// SIMATIC S7-200 project (STEP 7-Micro/WIN), CPU 224 REL 02.01

SYMBOL_TABLE USER1
Wazn_HMI         VW228
Meghdare_rikhteshode_hm VW226
Timer_for_not_reset_CNT T111
Time_for_stop_tow T110
Reset_Tow_HMI    V152.7
Overload_Feeder  I2.7
Counter_tow      C10
Metraj_Mohasebe_shod VW224
wazn1            VW232
NM               VW230
ktex             VW222
Wazn_mored_niaz  VW220
Start_motor_water_mod V152.5
Start_motor      V152.4
SQ_Press         I0.0     // Sensore roye jack dar moghiyate press
SQ_Watter        I0.1     // Sensore roye jack dar moghiyate abgiri
SQ_Front         I0.2     // Sensore roye jacke taghziye  dar moghiyate jelo
SQ_Back          I0.3     // Sensore roye jacke taghziye  dar moghiyate aghab
Level            I0.4     // farmane level control
Start_Press      I0.5     // kelide start marboot be amaliate press
Start_Watter     I0.6     // kelide start marboot be amaliate abgiri
Stopp            I0.7     // kelide Stop
Emergency        I1.0     // Emergency
SQ_Up_Press      I1.1     // Sensore elghaei jahate tashkhise balabodane press
Pressure_SW      I1.2     // perssure switch_farmane paein raftane peres ra ghat mikonad
Overload_Mainmotor I1.3     // Overload
Overload_Pump    I1.4     // Overload
Sensor_Tow       I1.5     // Overload
SQ_Down_Press    I2.0     // Sensore elghaei jahate tashkhise paein bodane press
SQ_Metraj        I2.1
SQ_12mm          I2.2     // sensore 12mm baghale sotun jahate tashkhise peres
SQ_pichesheKats  I2.3     // Picheshe Kats
Motor_Pump       Q0.0     // Watter Pump
Motor_Feeder     Q0.1     // Feeder Motor
EV_H_Mot         Q0.2     // valve hidrolik for hidromotor
EV_H_Press_Up    Q0.3     // valve hidrolik press go to up
EV_H_Press_Down  Q0.4     // valve hidrolik press go to down
EV_J_Press       Q0.5     // shir barghi jak baraye raftan be moghiyate press
EV_J_Water       Q0.6     // shir barghi jak baraye raftan be moghiyate abgiri
EV_J_Forward     Q0.7     // shirbarghi  jak baraye raftan be moghiyate taghziye dadan
EV_J_Backward    Q1.0     // shirbarghi  jak baraye raftan be moghiyate aghab
Contactor_Main   Q1.1     // Contactor_Main (Motore Hidrolik)
Contactor_Star   Q2.0     // Contactor_Star (Motore Hidrolik)
Contactor_Delta  Q2.1     // Contactor_Delta (Motore Hidrolik)
Stream           Q2.2     // shire Bokhar
Watter           Q2.3     // shire aab
Drive_Kats       Q2.4     // Kats
MainValve        Q2.5
Safty_Timer      T37
Machin_Fault     V100.0
Fault_MainMotor  V100.1
Fault_MotorPUMP  V100.2
Fault_Feeder     V100.3
Finish_watter    V100.4
Manual           V100.5
Finish_press     V100.6
Flag4            V100.7
Mainmotor_on_HMI V101.0
Flag1            V101.1
Flag2            V101.2
Flag3            V101.3
Flag1_w          V101.4
Flag2_w          V101.5
Flag_water1      V101.6
Reset_C1         V101.7
reset_c2         V102.0
manual_move_feeder V102.1
Start_watter_hmi V151.0
Start_press_hmi  V151.1   // dokmeye start peress dar HMI
H_Motor_hmi      V151.2
W_Motor_hmi      V151.3
F_Motor_hmi      V151.4
Press_up_hmi     V151.5
Press_down_hmi   V151.6
jack_press_hmi   V151.7
Jack_watter_hmi  V152.0
Jack_feeder_Front_hmi V152.1
Jack_feeder_Back_hmi V152.2
drive_manual_hmi V152.3
Temperatur       VD800
Enable_Stream    VW200
Setpoint_Temp    VW202
Enable_Watter_hmi VW204
Metraj           VW206
time_press       VW208
meghdare_counter1 VW210
END_SYMBOL_TABLE

ORGANIZATION_BLOCK MAIN:OB1
TITLE=[v100- v110--->bit] , [ V110-V150 ]---->Retentive
// [v151-v161]--->bit  , [ V151-V199 ]
// -----------------------------------------------------------------
// [ VW200-VW398]---->Retentive
// [ VW400-VW598]
// -----------------------------------------------------------------
// [ VD600-VD796 ]---->Retentive
// [ VD800- ^|^    ]
// -----------------------------------------------------------------
// [ T37-T40 ]---->Retentive
// 
BEGIN
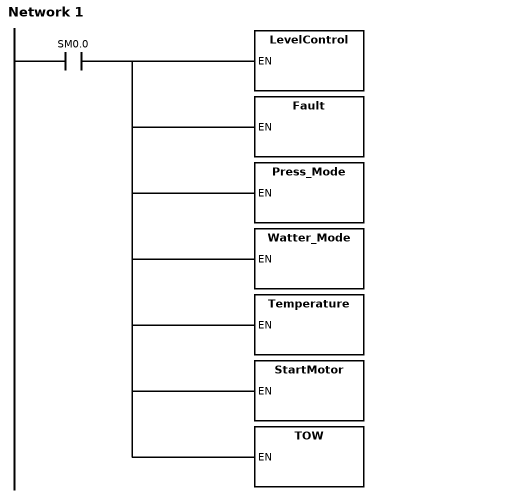
Network 1
LD     SM0.0
CALL   LevelControl:SBR0
CALL   Fault:SBR1
CALL   Press_Mode:SBR2
CALL   Watter_Mode:SBR3
CALL   Temperature:SBR4
CALL   StartMotor:SBR5
CALL   TOW:SBR6
END_ORGANIZATION_BLOCK

SUBROUTINE_BLOCK LevelControl:SBR0
TITLE=SUBROUTINE COMMENTS
BEGIN
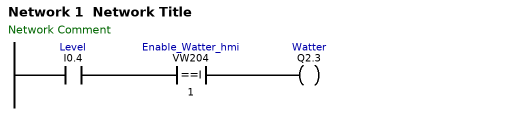
Network 1 // Network Title
// Network Comment
LD     Level:I0.4
AW=    Enable_Watter_hmi:VW204, 1
=      Watter:Q2.3
END_SUBROUTINE_BLOCK

SUBROUTINE_BLOCK Fault:SBR1
TITLE=SUBROUTINE COMMENTS
BEGIN
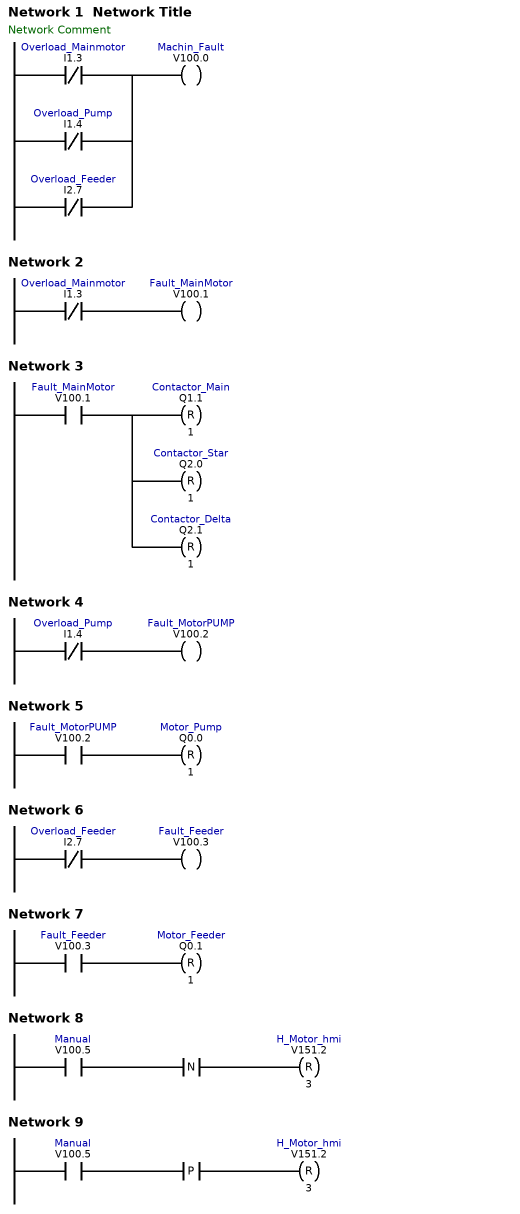
Network 1 // Network Title
// Network Comment
LDN    Overload_Mainmotor:I1.3
ON     Overload_Pump:I1.4
ON     Overload_Feeder:I2.7
=      Machin_Fault:V100.0
Network 2
LDN    Overload_Mainmotor:I1.3
=      Fault_MainMotor:V100.1
Network 3
LD     Fault_MainMotor:V100.1
R      Contactor_Main:Q1.1, 1
R      Contactor_Star:Q2.0, 1
R      Contactor_Delta:Q2.1, 1
Network 4
LDN    Overload_Pump:I1.4
=      Fault_MotorPUMP:V100.2
Network 5
LD     Fault_MotorPUMP:V100.2
R      Motor_Pump:Q0.0, 1
Network 6
LDN    Overload_Feeder:I2.7
=      Fault_Feeder:V100.3
Network 7
LD     Fault_Feeder:V100.3
R      Motor_Feeder:Q0.1, 1
Network 8
LD     Manual:V100.5
ED
R      H_Motor_hmi:V151.2, 3
Network 9
LD     Manual:V100.5
EU
R      H_Motor_hmi:V151.2, 3
END_SUBROUTINE_BLOCK

SUBROUTINE_BLOCK Press_Mode:SBR2
TITLE=SUBROUTINE COMMENTS
BEGIN
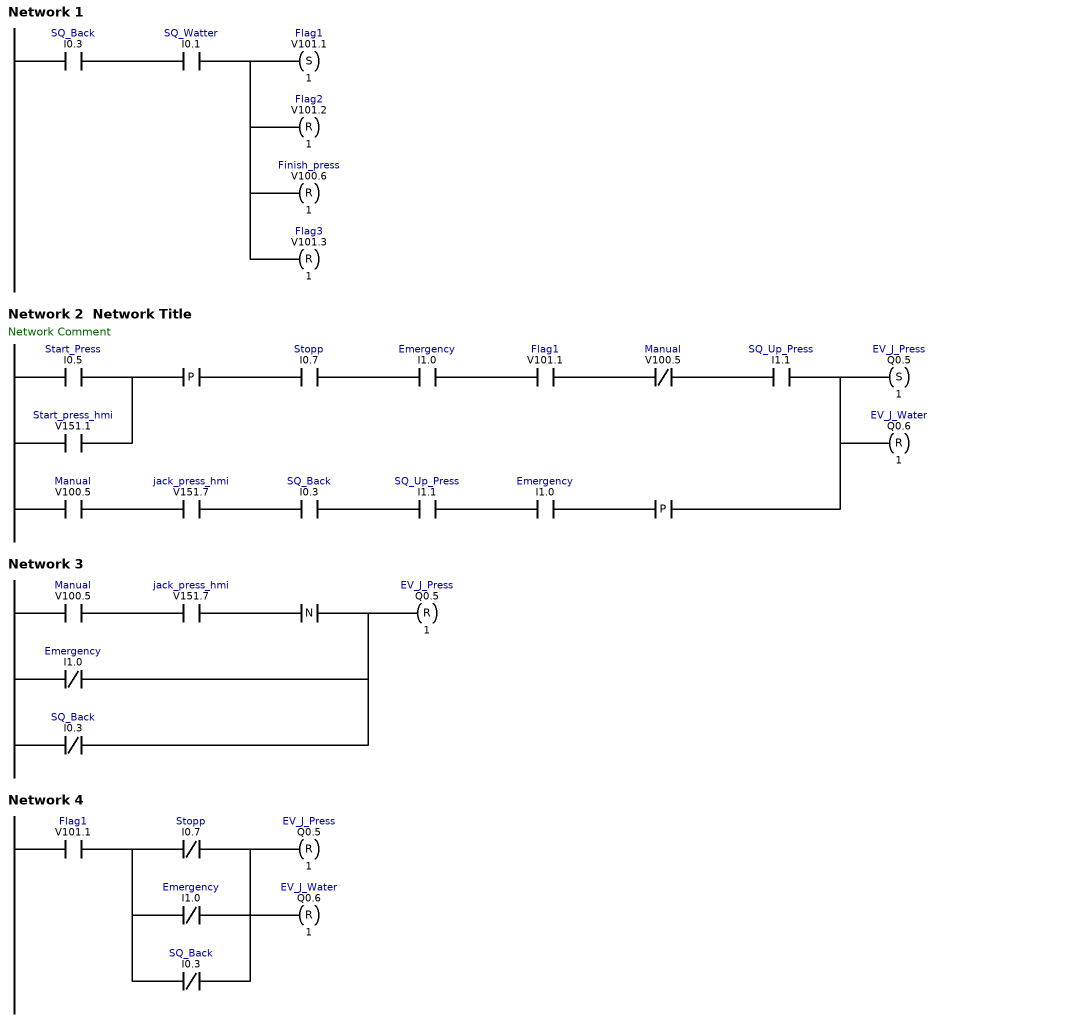
Network 1
LD     SQ_Back:I0.3
A      SQ_Watter:I0.1
S      Flag1:V101.1, 1
R      Flag2:V101.2, 1
R      Finish_press:V100.6, 1
R      Flag3:V101.3, 1
Network 2 // Network Title
// Network Comment
LD     Start_Press:I0.5
O      Start_press_hmi:V151.1
EU
A      Stopp:I0.7
A      Emergency:I1.0
A      Flag1:V101.1
AN     Manual:V100.5
A      SQ_Up_Press:I1.1
LD     Manual:V100.5
A      jack_press_hmi:V151.7
A      SQ_Back:I0.3
A      SQ_Up_Press:I1.1
A      Emergency:I1.0
EU
OLD
S      EV_J_Press:Q0.5, 1
R      EV_J_Water:Q0.6, 1
Network 3
LD     Manual:V100.5
A      jack_press_hmi:V151.7
ED
ON     Emergency:I1.0
ON     SQ_Back:I0.3
R      EV_J_Press:Q0.5, 1
Network 4
LD     Flag1:V101.1
LDN    Stopp:I0.7
ON     Emergency:I1.0
ON     SQ_Back:I0.3
ALD
R      EV_J_Press:Q0.5, 1
R      EV_J_Water:Q0.6, 1
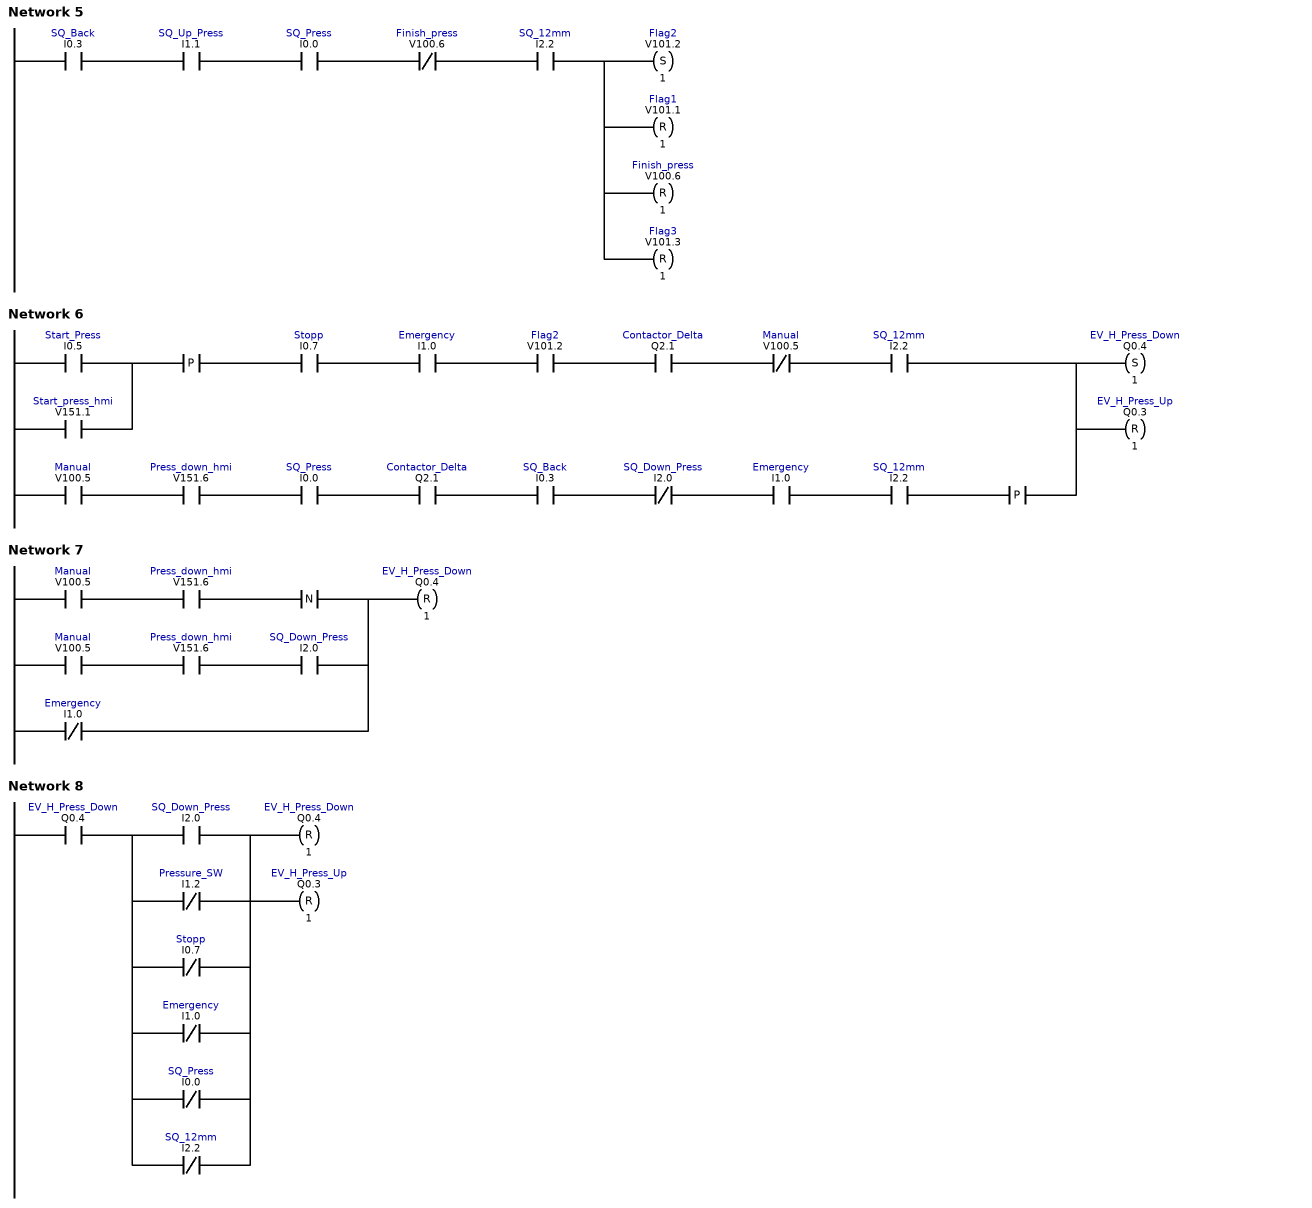
Network 5
LD     SQ_Back:I0.3
A      SQ_Up_Press:I1.1
A      SQ_Press:I0.0
AN     Finish_press:V100.6
A      SQ_12mm:I2.2
S      Flag2:V101.2, 1
R      Flag1:V101.1, 1
R      Finish_press:V100.6, 1
R      Flag3:V101.3, 1
Network 6
LD     Start_Press:I0.5
O      Start_press_hmi:V151.1
EU
A      Stopp:I0.7
A      Emergency:I1.0
A      Flag2:V101.2
A      Contactor_Delta:Q2.1
AN     Manual:V100.5
A      SQ_12mm:I2.2
LD     Manual:V100.5
A      Press_down_hmi:V151.6
A      SQ_Press:I0.0
A      Contactor_Delta:Q2.1
A      SQ_Back:I0.3
AN     SQ_Down_Press:I2.0
A      Emergency:I1.0
A      SQ_12mm:I2.2
EU
OLD
S      EV_H_Press_Down:Q0.4, 1
R      EV_H_Press_Up:Q0.3, 1
Network 7
LD     Manual:V100.5
A      Press_down_hmi:V151.6
ED
LD     Manual:V100.5
A      Press_down_hmi:V151.6
A      SQ_Down_Press:I2.0
OLD
ON     Emergency:I1.0
R      EV_H_Press_Down:Q0.4, 1
Network 8
LD     EV_H_Press_Down:Q0.4
LD     SQ_Down_Press:I2.0
ON     Pressure_SW:I1.2
ON     Stopp:I0.7
ON     Emergency:I1.0
ON     SQ_Press:I0.0
ON     SQ_12mm:I2.2
ALD
R      EV_H_Press_Down:Q0.4, 1
R      EV_H_Press_Up:Q0.3, 1
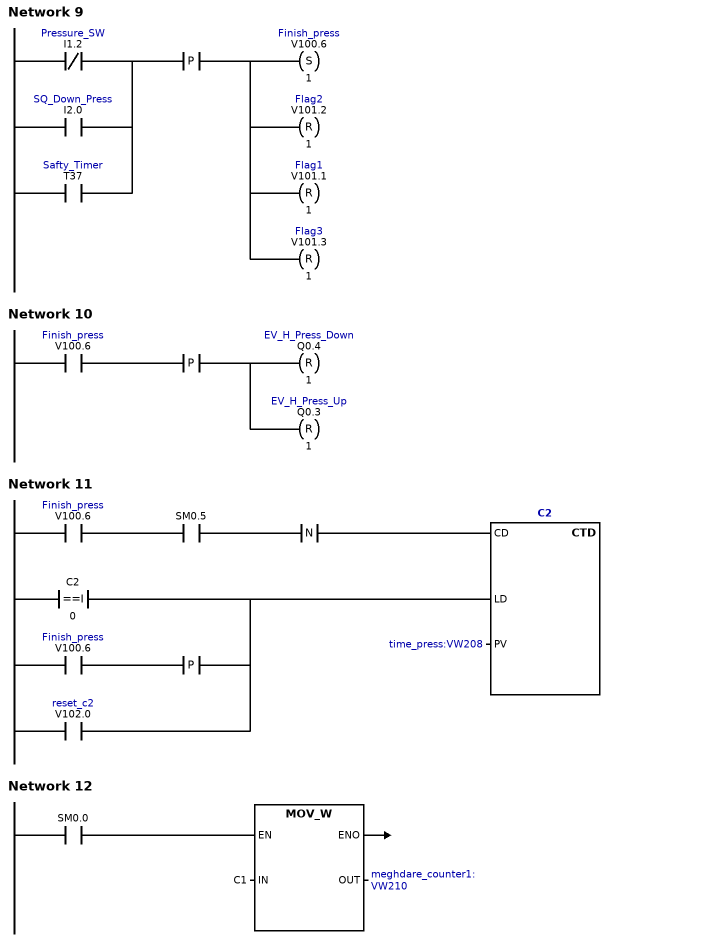
Network 9
LDN    Pressure_SW:I1.2
O      SQ_Down_Press:I2.0
O      Safty_Timer:T37
EU
S      Finish_press:V100.6, 1
R      Flag2:V101.2, 1
R      Flag1:V101.1, 1
R      Flag3:V101.3, 1
Network 10
LD     Finish_press:V100.6
EU
R      EV_H_Press_Down:Q0.4, 1
R      EV_H_Press_Up:Q0.3, 1
Network 11
LD     Finish_press:V100.6
A      SM0.5
ED
LDW=   C2, 0
LD     Finish_press:V100.6
EU
OLD
O      reset_c2:V102.0
CTD    C2, time_press:VW208
Network 12
LD     SM0.0
MOVW   C1, meghdare_counter1:VW210
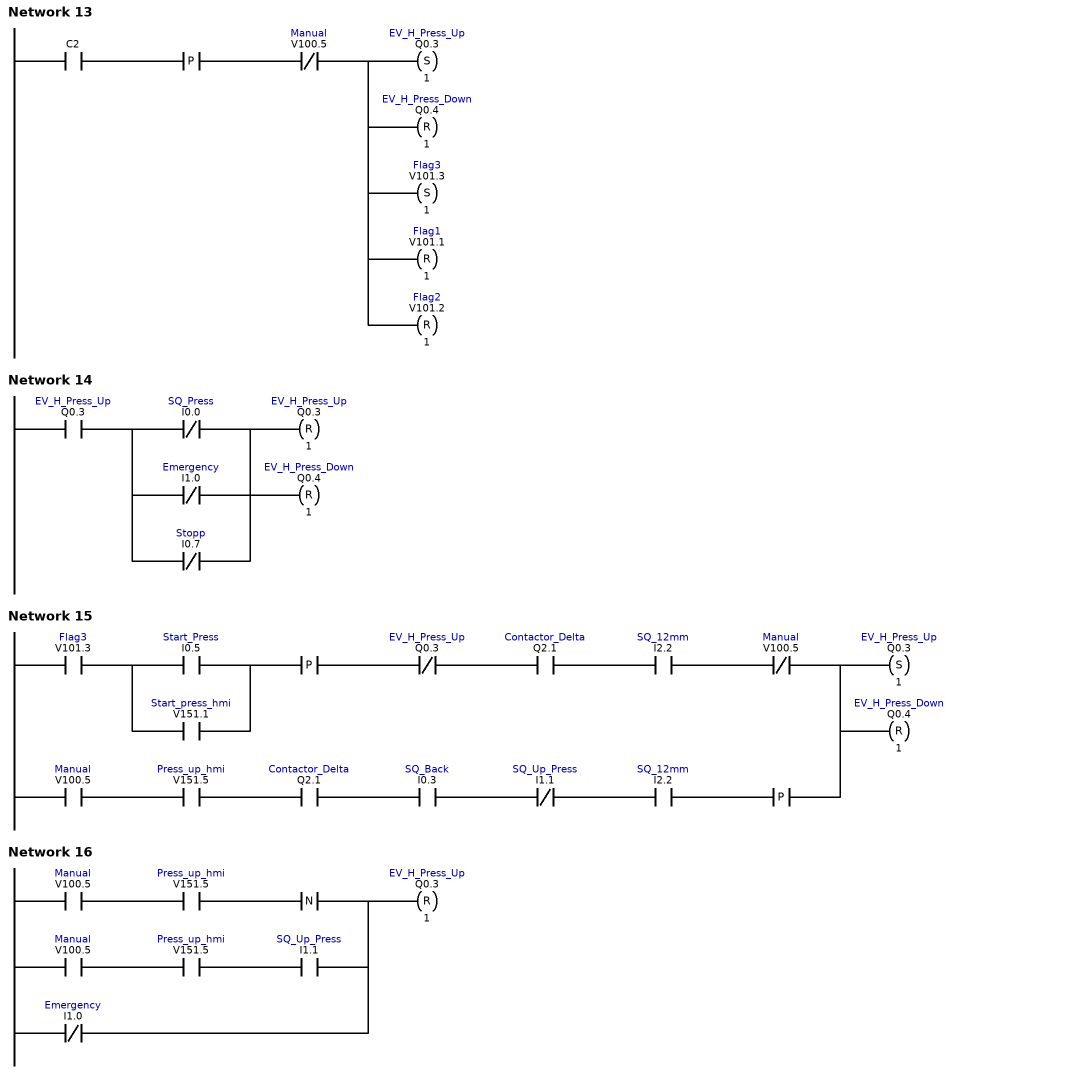
Network 13
LD     C2
EU
AN     Manual:V100.5
S      EV_H_Press_Up:Q0.3, 1
R      EV_H_Press_Down:Q0.4, 1
S      Flag3:V101.3, 1
R      Flag1:V101.1, 1
R      Flag2:V101.2, 1
Network 14
LD     EV_H_Press_Up:Q0.3
LDN    SQ_Press:I0.0
ON     Emergency:I1.0
ON     Stopp:I0.7
ALD
R      EV_H_Press_Up:Q0.3, 1
R      EV_H_Press_Down:Q0.4, 1
Network 15
LD     Flag3:V101.3
LD     Start_Press:I0.5
O      Start_press_hmi:V151.1
ALD
EU
AN     EV_H_Press_Up:Q0.3
A      Contactor_Delta:Q2.1
A      SQ_12mm:I2.2
AN     Manual:V100.5
LD     Manual:V100.5
A      Press_up_hmi:V151.5
A      Contactor_Delta:Q2.1
A      SQ_Back:I0.3
AN     SQ_Up_Press:I1.1
A      SQ_12mm:I2.2
EU
OLD
S      EV_H_Press_Up:Q0.3, 1
R      EV_H_Press_Down:Q0.4, 1
Network 16
LD     Manual:V100.5
A      Press_up_hmi:V151.5
ED
LD     Manual:V100.5
A      Press_up_hmi:V151.5
A      SQ_Up_Press:I1.1
OLD
ON     Emergency:I1.0
R      EV_H_Press_Up:Q0.3, 1
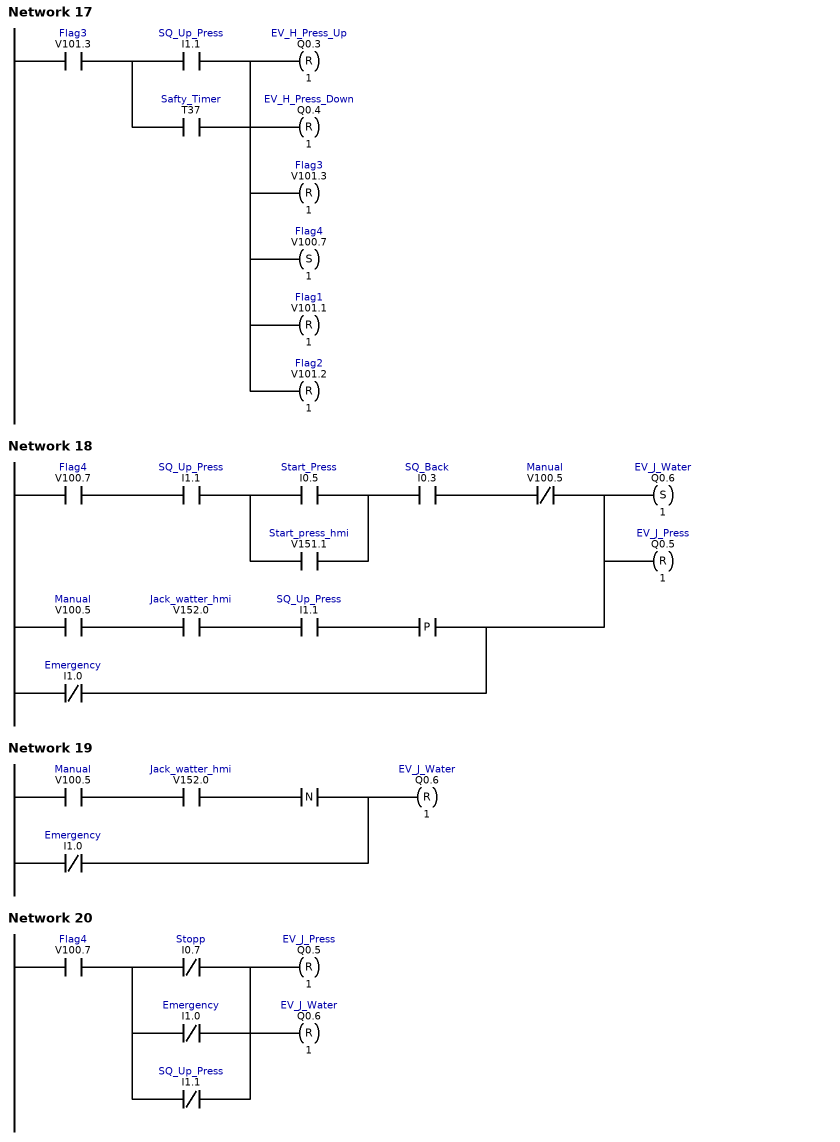
Network 17
LD     Flag3:V101.3
LD     SQ_Up_Press:I1.1
O      Safty_Timer:T37
ALD
R      EV_H_Press_Up:Q0.3, 1
R      EV_H_Press_Down:Q0.4, 1
R      Flag3:V101.3, 1
S      Flag4:V100.7, 1
R      Flag1:V101.1, 1
R      Flag2:V101.2, 1
Network 18
LD     Flag4:V100.7
A      SQ_Up_Press:I1.1
LD     Start_Press:I0.5
O      Start_press_hmi:V151.1
ALD
A      SQ_Back:I0.3
AN     Manual:V100.5
LD     Manual:V100.5
A      Jack_watter_hmi:V152.0
A      SQ_Up_Press:I1.1
EU
ON     Emergency:I1.0
OLD
S      EV_J_Water:Q0.6, 1
R      EV_J_Press:Q0.5, 1
Network 19
LD     Manual:V100.5
A      Jack_watter_hmi:V152.0
ED
ON     Emergency:I1.0
R      EV_J_Water:Q0.6, 1
Network 20
LD     Flag4:V100.7
LDN    Stopp:I0.7
ON     Emergency:I1.0
ON     SQ_Up_Press:I1.1
ALD
R      EV_J_Press:Q0.5, 1
R      EV_J_Water:Q0.6, 1
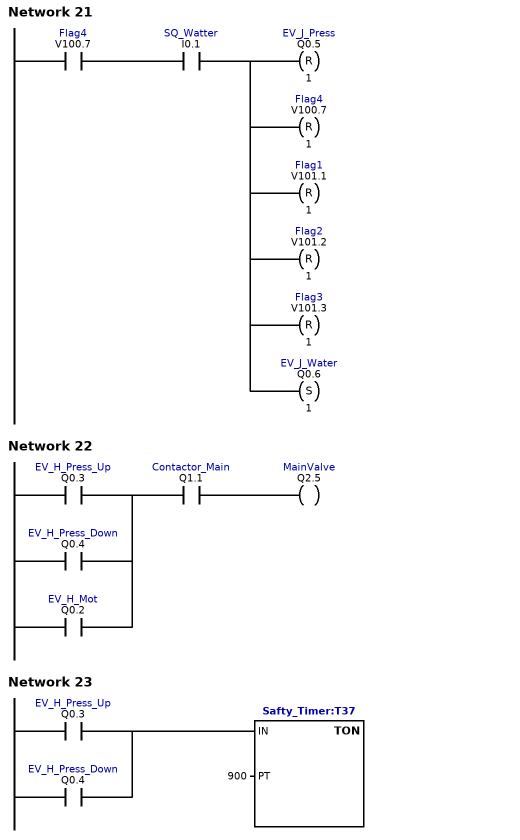
Network 21
LD     Flag4:V100.7
A      SQ_Watter:I0.1
R      EV_J_Press:Q0.5, 1
R      Flag4:V100.7, 1
R      Flag1:V101.1, 1
R      Flag2:V101.2, 1
R      Flag3:V101.3, 1
S      EV_J_Water:Q0.6, 1
Network 22
LD     EV_H_Press_Up:Q0.3
O      EV_H_Press_Down:Q0.4
O      EV_H_Mot:Q0.2
A      Contactor_Main:Q1.1
=      MainValve:Q2.5
Network 23
LD     EV_H_Press_Up:Q0.3
O      EV_H_Press_Down:Q0.4
TON    Safty_Timer:T37, 900
END_SUBROUTINE_BLOCK

SUBROUTINE_BLOCK Watter_Mode:SBR3
TITLE=SUBROUTINE COMMENTS
VAR
metraj1:INT;	// LW0 
metraj2:INT;	// LW2 
out:BOOL;	// L4.0 
END_VAR
BEGIN
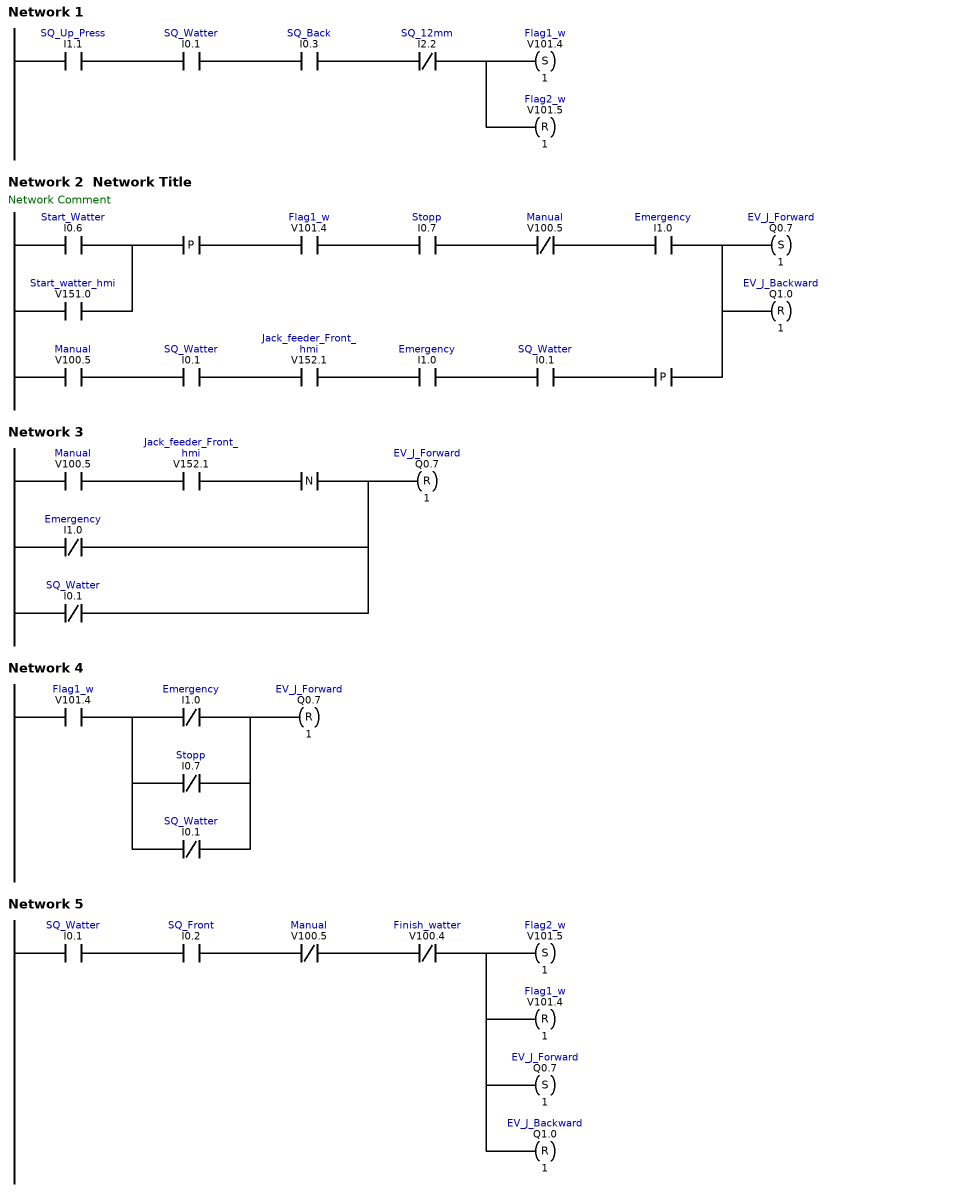
Network 1
LD     SQ_Up_Press:I1.1
A      SQ_Watter:I0.1
A      SQ_Back:I0.3
AN     SQ_12mm:I2.2
S      Flag1_w:V101.4, 1
R      Flag2_w:V101.5, 1
Network 2 // Network Title
// Network Comment
LD     Start_Watter:I0.6
O      Start_watter_hmi:V151.0
EU
A      Flag1_w:V101.4
A      Stopp:I0.7
AN     Manual:V100.5
A      Emergency:I1.0
LD     Manual:V100.5
A      SQ_Watter:I0.1
A      Jack_feeder_Front_hmi:V152.1
A      Emergency:I1.0
A      SQ_Watter:I0.1
EU
OLD
S      EV_J_Forward:Q0.7, 1
R      EV_J_Backward:Q1.0, 1
Network 3
LD     Manual:V100.5
A      Jack_feeder_Front_hmi:V152.1
ED
ON     Emergency:I1.0
ON     SQ_Watter:I0.1
R      EV_J_Forward:Q0.7, 1
Network 4
LD     Flag1_w:V101.4
LDN    Emergency:I1.0
ON     Stopp:I0.7
ON     SQ_Watter:I0.1
ALD
R      EV_J_Forward:Q0.7, 1
Network 5
LD     SQ_Watter:I0.1
A      SQ_Front:I0.2
AN     Manual:V100.5
AN     Finish_watter:V100.4
S      Flag2_w:V101.5, 1
R      Flag1_w:V101.4, 1
S      EV_J_Forward:Q0.7, 1
R      EV_J_Backward:Q1.0, 1
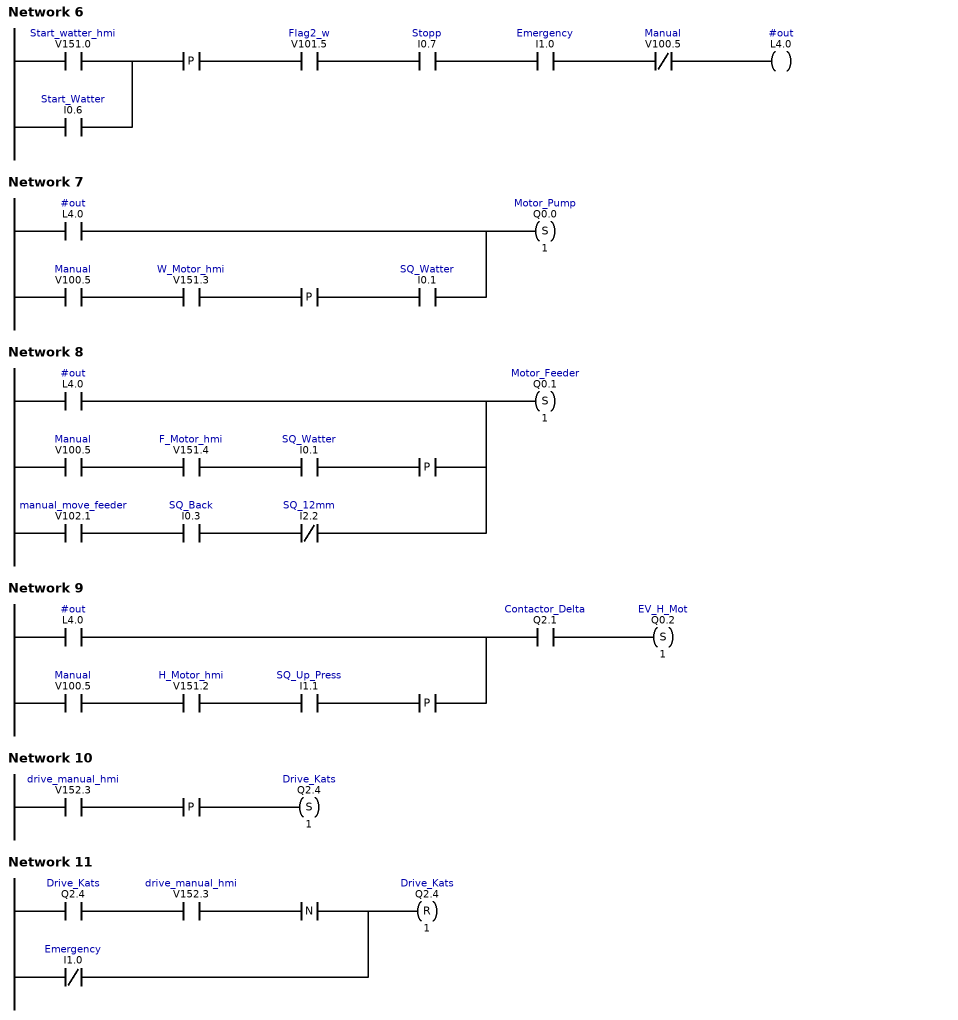
Network 6
LD     Start_watter_hmi:V151.0
O      Start_Watter:I0.6
EU
A      Flag2_w:V101.5
A      Stopp:I0.7
A      Emergency:I1.0
AN     Manual:V100.5
=      #out:L4.0
Network 7
LD     #out:L4.0
LD     Manual:V100.5
A      W_Motor_hmi:V151.3
EU
A      SQ_Watter:I0.1
OLD
S      Motor_Pump:Q0.0, 1
Network 8
LD     #out:L4.0
LD     Manual:V100.5
A      F_Motor_hmi:V151.4
A      SQ_Watter:I0.1
EU
OLD
LD     manual_move_feeder:V102.1
A      SQ_Back:I0.3
AN     SQ_12mm:I2.2
OLD
S      Motor_Feeder:Q0.1, 1
Network 9
LD     #out:L4.0
LD     Manual:V100.5
A      H_Motor_hmi:V151.2
A      SQ_Up_Press:I1.1
EU
OLD
A      Contactor_Delta:Q2.1
S      EV_H_Mot:Q0.2, 1
Network 10
LD     drive_manual_hmi:V152.3
EU
S      Drive_Kats:Q2.4, 1
Network 11
LD     Drive_Kats:Q2.4
A      drive_manual_hmi:V152.3
ED
ON     Emergency:I1.0
R      Drive_Kats:Q2.4, 1
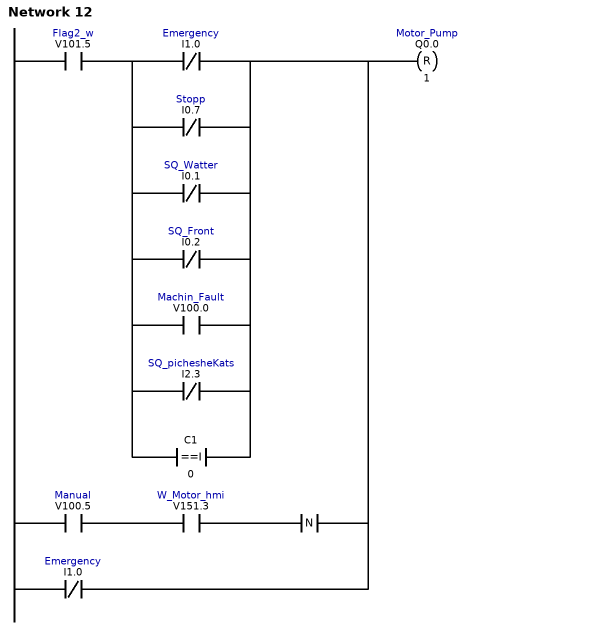
Network 12
LD     Flag2_w:V101.5
LDN    Emergency:I1.0
ON     Stopp:I0.7
ON     SQ_Watter:I0.1
ON     SQ_Front:I0.2
O      Machin_Fault:V100.0
ON     SQ_pichesheKats:I2.3
OW=    C1, 0
ALD
LD     Manual:V100.5
A      W_Motor_hmi:V151.3
ED
ON     Emergency:I1.0
OLD
R      Motor_Pump:Q0.0, 1
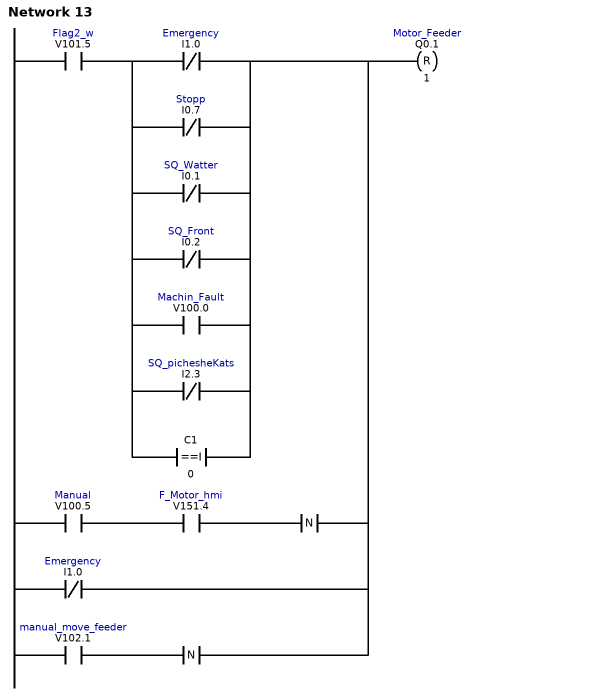
Network 13
LD     Flag2_w:V101.5
LDN    Emergency:I1.0
ON     Stopp:I0.7
ON     SQ_Watter:I0.1
ON     SQ_Front:I0.2
O      Machin_Fault:V100.0
ON     SQ_pichesheKats:I2.3
OW=    C1, 0
ALD
LD     Manual:V100.5
A      F_Motor_hmi:V151.4
ED
ON     Emergency:I1.0
LD     manual_move_feeder:V102.1
ED
OLD
OLD
R      Motor_Feeder:Q0.1, 1
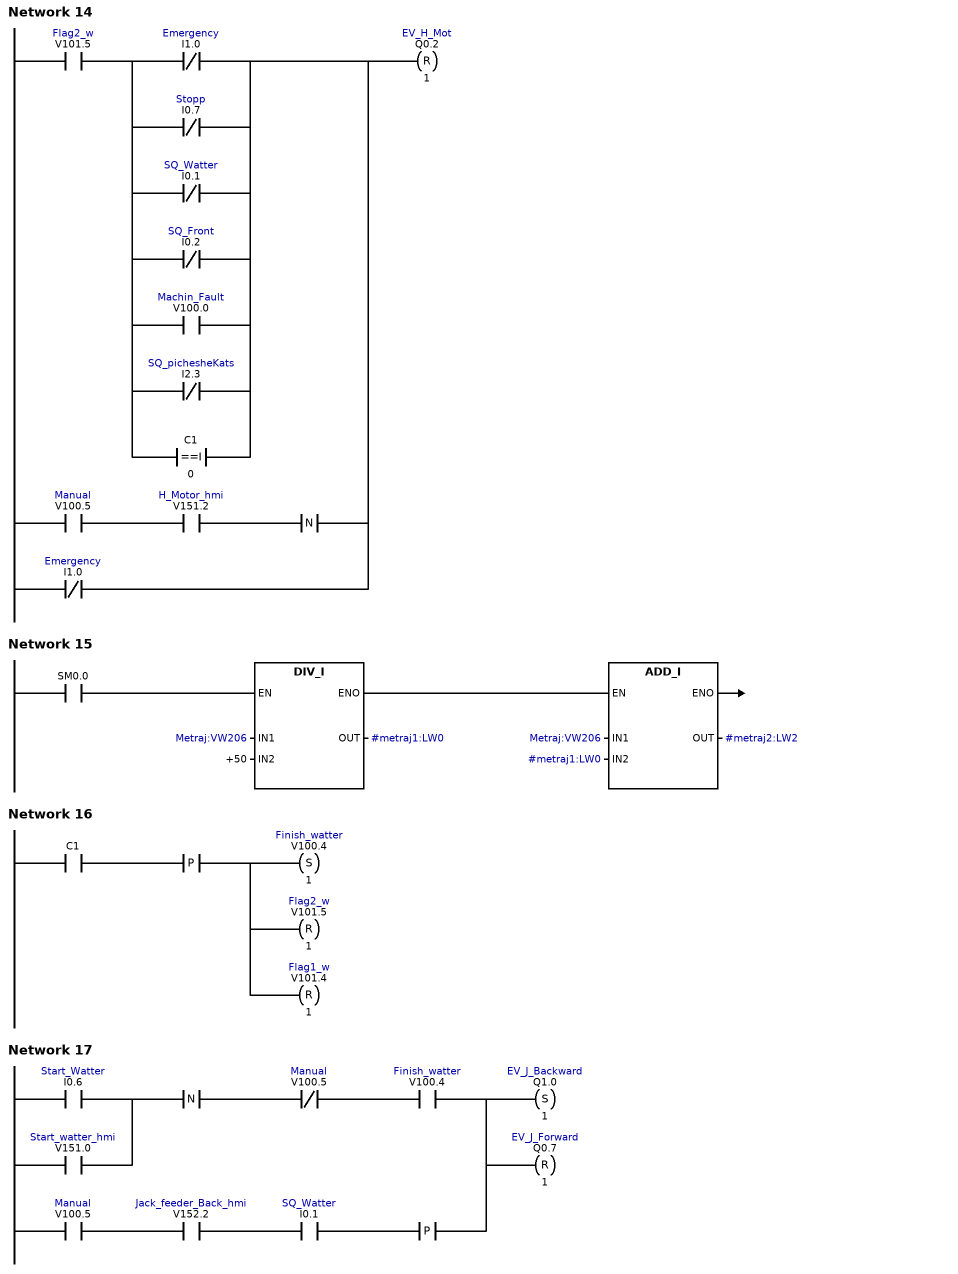
Network 14
LD     Flag2_w:V101.5
LDN    Emergency:I1.0
ON     Stopp:I0.7
ON     SQ_Watter:I0.1
ON     SQ_Front:I0.2
O      Machin_Fault:V100.0
ON     SQ_pichesheKats:I2.3
OW=    C1, 0
ALD
LD     Manual:V100.5
A      H_Motor_hmi:V151.2
ED
ON     Emergency:I1.0
OLD
R      EV_H_Mot:Q0.2, 1
Network 15
LD     SM0.0
MOVW   Metraj:VW206, #metraj1:LW0
AENO
/I     +50, #metraj1:LW0
AENO
MOVW   Metraj:VW206, #metraj2:LW2
+I     #metraj1:LW0, #metraj2:LW2
Network 16
LD     C1
EU
S      Finish_watter:V100.4, 1
R      Flag2_w:V101.5, 1
R      Flag1_w:V101.4, 1
Network 17
LD     Start_Watter:I0.6
O      Start_watter_hmi:V151.0
ED
AN     Manual:V100.5
A      Finish_watter:V100.4
LD     Manual:V100.5
A      Jack_feeder_Back_hmi:V152.2
A      SQ_Watter:I0.1
EU
OLD
S      EV_J_Backward:Q1.0, 1
R      EV_J_Forward:Q0.7, 1
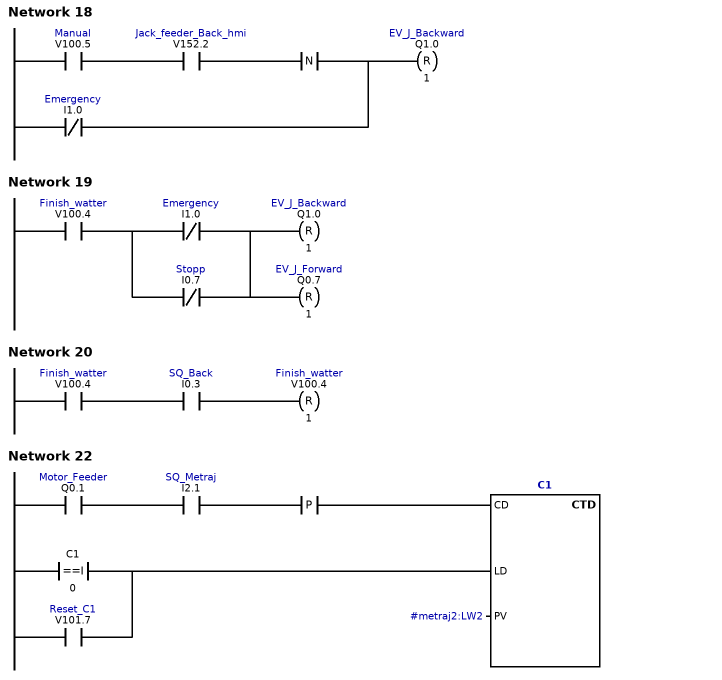
Network 18
LD     Manual:V100.5
A      Jack_feeder_Back_hmi:V152.2
ED
ON     Emergency:I1.0
R      EV_J_Backward:Q1.0, 1
Network 19
LD     Finish_watter:V100.4
LDN    Emergency:I1.0
ON     Stopp:I0.7
ALD
R      EV_J_Backward:Q1.0, 1
R      EV_J_Forward:Q0.7, 1
Network 20
LD     Finish_watter:V100.4
A      SQ_Back:I0.3
R      Finish_watter:V100.4, 1
Network 22
LD     Motor_Feeder:Q0.1
A      SQ_Metraj:I2.1
EU
LDW=   C1, 0
O      Reset_C1:V101.7
CTD    C1, #metraj2:LW2
END_SUBROUTINE_BLOCK

SUBROUTINE_BLOCK Temperature:SBR4
TITLE=SUBROUTINE COMMENTS
VAR
Dama1:WORD;	// LW0 
Dama2:DWORD;	// LD2 
Dama3:REAL;	// LD6 
Dama4:REAL;	// LD10 
Dama:REAL;	// LD14 damaye vaghei
Dama_Round1:DINT;	// LD18 damaye round shode_DIN
Dama_Round:INT;	// LW22 damaye round shode_IN
Dama_Round_2:INT;	// LW24 setpoint-2
dama_10:INT;	// LW26 
END_VAR
BEGIN
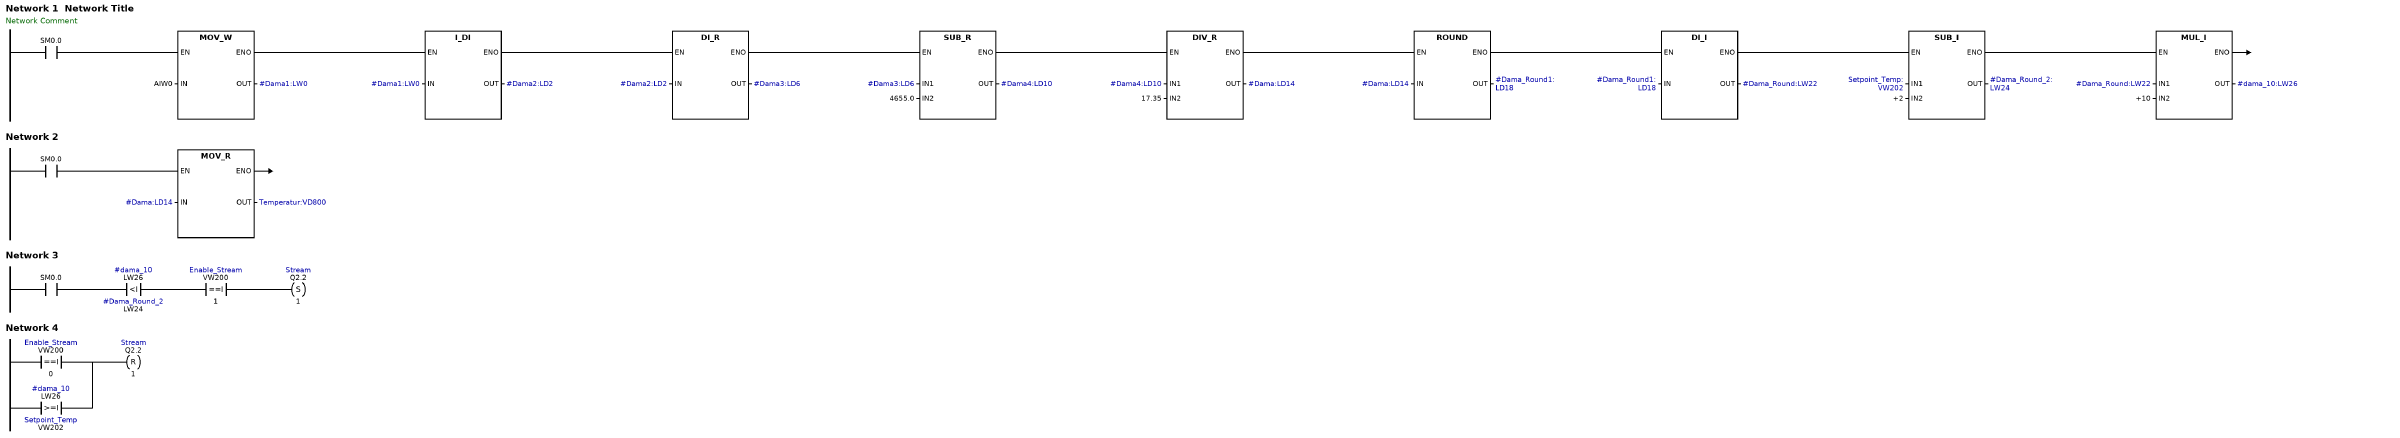
Network 1 // Network Title
// Network Comment
LD     SM0.0
MOVW   AIW0, #Dama1:LW0
AENO
ITD    #Dama1:LW0, #Dama2:LD2
AENO
DTR    #Dama2:LD2, #Dama3:LD6
AENO
MOVR   #Dama3:LD6, #Dama4:LD10
AENO
-R     4655.0, #Dama4:LD10
AENO
MOVR   #Dama4:LD10, #Dama:LD14
AENO
/R     17.35, #Dama:LD14
AENO
ROUND  #Dama:LD14, #Dama_Round1:LD18
AENO
DTI    #Dama_Round1:LD18, #Dama_Round:LW22
AENO
MOVW   Setpoint_Temp:VW202, #Dama_Round_2:LW24
AENO
-I     +2, #Dama_Round_2:LW24
AENO
MOVW   #Dama_Round:LW22, #dama_10:LW26
*I     +10, #dama_10:LW26
Network 2
LD     SM0.0
MOVR   #Dama:LD14, Temperatur:VD800
Network 3
LD     SM0.0
AW<    #dama_10:LW26, #Dama_Round_2:LW24
AW=    Enable_Stream:VW200, 1
S      Stream:Q2.2, 1
Network 4
//  
LDW=   Enable_Stream:VW200, 0
OW>=   #dama_10:LW26, Setpoint_Temp:VW202
R      Stream:Q2.2, 1
END_SUBROUTINE_BLOCK

SUBROUTINE_BLOCK StartMotor:SBR5
TITLE=SUBROUTINE COMMENTS
BEGIN
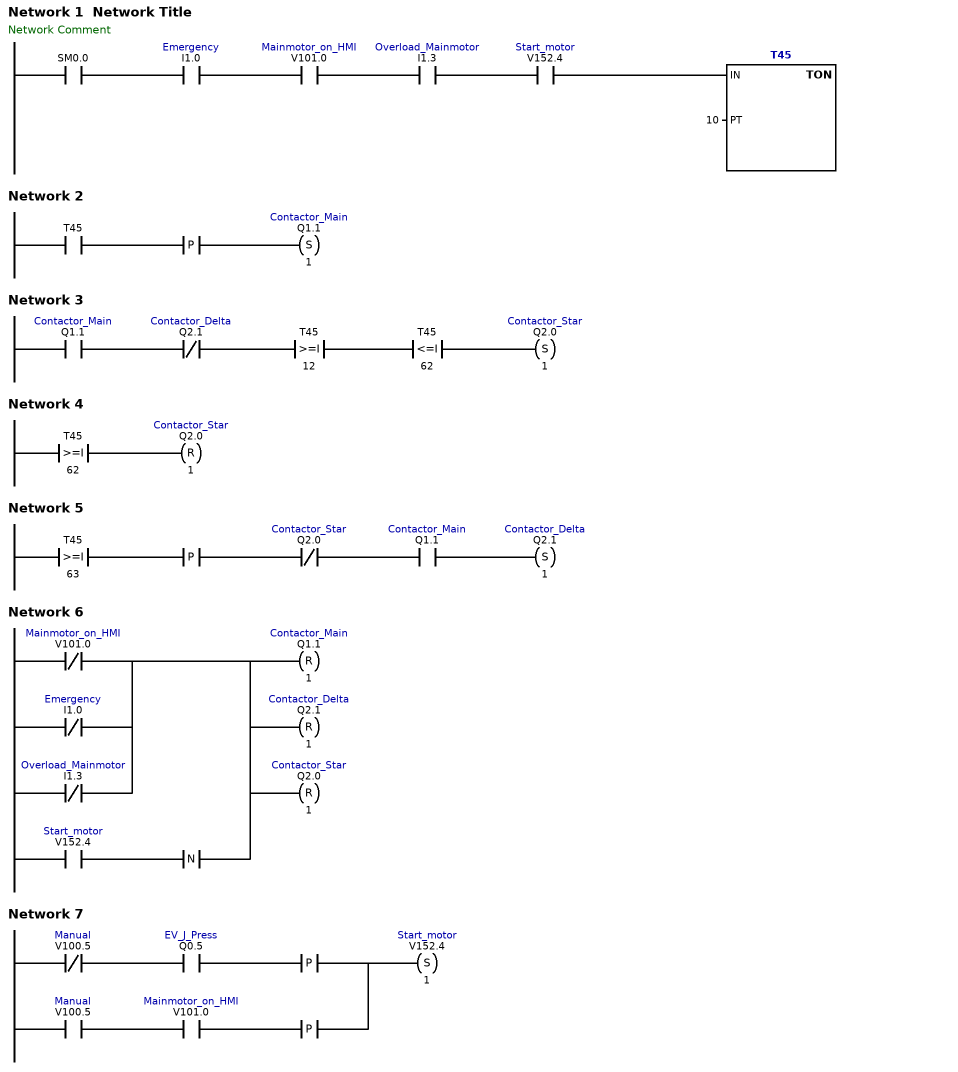
Network 1 // Network Title
// Network Comment
LD     SM0.0
A      Emergency:I1.0
A      Mainmotor_on_HMI:V101.0
A      Overload_Mainmotor:I1.3
A      Start_motor:V152.4
TON    T45, 10
Network 2
LD     T45
EU
S      Contactor_Main:Q1.1, 1
Network 3
LD     Contactor_Main:Q1.1
AN     Contactor_Delta:Q2.1
AW>=   T45, 12
AW<=   T45, 62
S      Contactor_Star:Q2.0, 1
Network 4
LDW>=  T45, 62
R      Contactor_Star:Q2.0, 1
Network 5
LDW>=  T45, 63
EU
AN     Contactor_Star:Q2.0
A      Contactor_Main:Q1.1
S      Contactor_Delta:Q2.1, 1
Network 6
LDN    Mainmotor_on_HMI:V101.0
ON     Emergency:I1.0
ON     Overload_Mainmotor:I1.3
LD     Start_motor:V152.4
ED
OLD
R      Contactor_Main:Q1.1, 1
R      Contactor_Delta:Q2.1, 1
R      Contactor_Star:Q2.0, 1
Network 7
LDN    Manual:V100.5
A      EV_J_Press:Q0.5
EU
LD     Manual:V100.5
A      Mainmotor_on_HMI:V101.0
EU
OLD
S      Start_motor:V152.4, 1
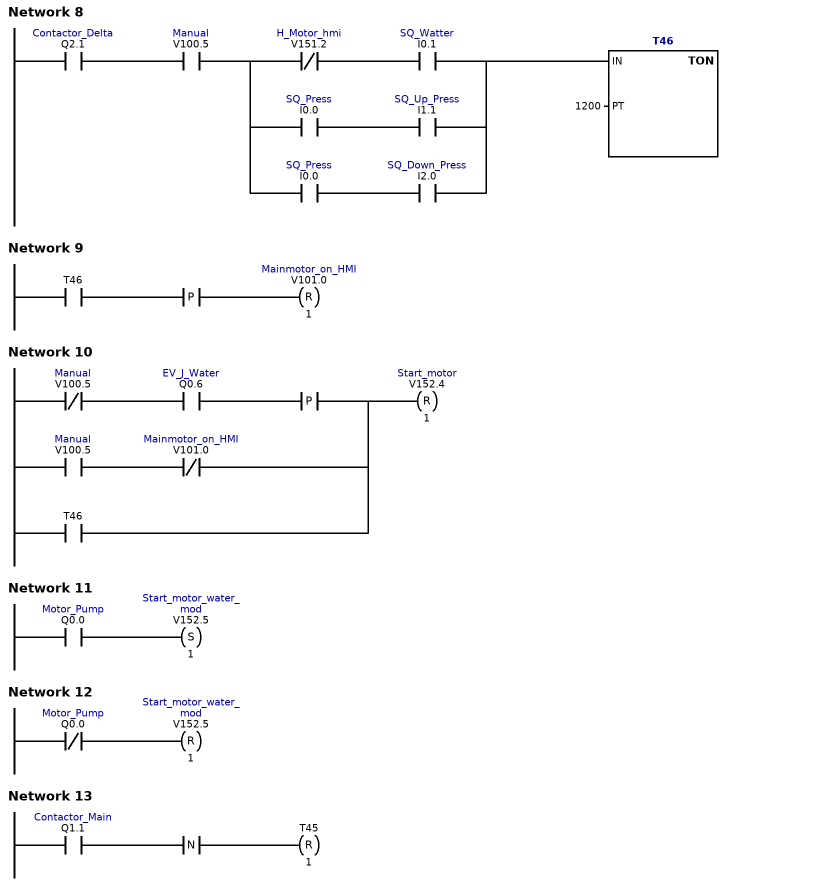
Network 8
LD     Contactor_Delta:Q2.1
A      Manual:V100.5
LDN    H_Motor_hmi:V151.2
A      SQ_Watter:I0.1
LD     SQ_Press:I0.0
A      SQ_Up_Press:I1.1
OLD
LD     SQ_Press:I0.0
A      SQ_Down_Press:I2.0
OLD
ALD
TON    T46, 1200
Network 9
LD     T46
EU
R      Mainmotor_on_HMI:V101.0, 1
Network 10
LDN    Manual:V100.5
A      EV_J_Water:Q0.6
EU
LD     Manual:V100.5
AN     Mainmotor_on_HMI:V101.0
OLD
O      T46
R      Start_motor:V152.4, 1
Network 11
LD     Motor_Pump:Q0.0
S      Start_motor_water_mod:V152.5, 1
Network 12
LDN    Motor_Pump:Q0.0
R      Start_motor_water_mod:V152.5, 1
Network 13
LD     Contactor_Main:Q1.1
ED
R      T45, 1
END_SUBROUTINE_BLOCK

SUBROUTINE_BLOCK TOW:SBR6
TITLE=INTERRUPT ROUTINE COMMENTS
VAR
metraj_Dword:DWORD;	// LD0 
metraj_cm:DWORD;	// LD4 
Tedade_dor:DWORD;	// LD8 
Tedade_dor_word:WORD;	// LW12 
Counter_DWord:DWORD;	// LD14 
cnt:DWORD;	// LD18 
metraje_rikhteshode_m:DWORD;	// LD22 
vazne_rikhte_shode:WORD;	// LW26 
NM_DW:DWORD;	// LD28 
wazn_DW:DWORD;	// LD32 
metraj_DW:DWORD;	// LD36 
metrajbar10:DWORD;	// LD40 
rikhteshode1:DWORD;	// LD44 
rikhteshode_DW:DWORD;	// LD48 
rikhteshode3:DWORD;	// LD52 
rikhte4:DWORD;	// LD56 
END_VAR
BEGIN
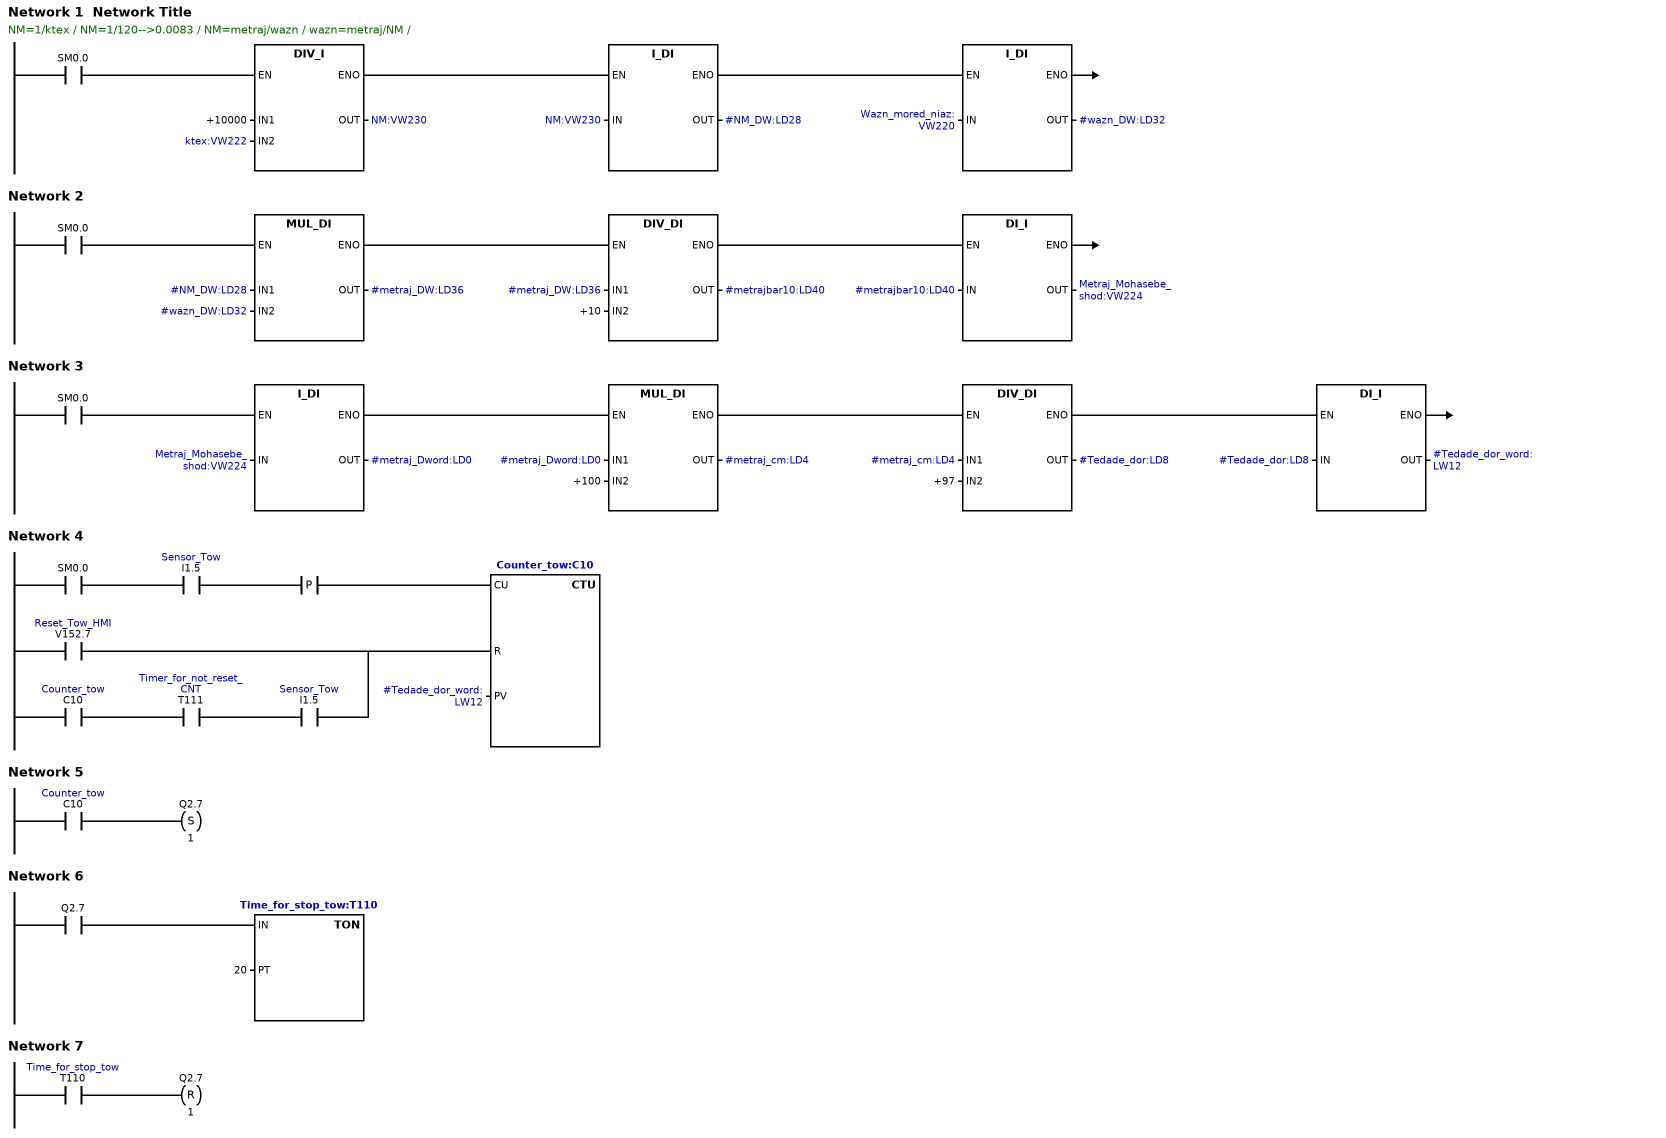
Network 1 // Network Title
// NM=1/ktex
// NM=1/120-->0.0083
// NM=metraj/wazn
// wazn=metraj/NM
// 
LD     SM0.0
MOVW   +10000, NM:VW230
AENO
/I     ktex:VW222, NM:VW230
AENO
ITD    NM:VW230, #NM_DW:LD28
AENO
ITD    Wazn_mored_niaz:VW220, #wazn_DW:LD32
Network 2
LD     SM0.0
MOVD   #NM_DW:LD28, #metraj_DW:LD36
AENO
*D     #wazn_DW:LD32, #metraj_DW:LD36
AENO
MOVD   #metraj_DW:LD36, #metrajbar10:LD40
AENO
/D     +10, #metrajbar10:LD40
AENO
DTI    #metrajbar10:LD40, Metraj_Mohasebe_shod:VW224
Network 3
LD     SM0.0
ITD    Metraj_Mohasebe_shod:VW224, #metraj_Dword:LD0
AENO
MOVD   #metraj_Dword:LD0, #metraj_cm:LD4
AENO
*D     +100, #metraj_cm:LD4
AENO
MOVD   #metraj_cm:LD4, #Tedade_dor:LD8
AENO
/D     +97, #Tedade_dor:LD8
AENO
DTI    #Tedade_dor:LD8, #Tedade_dor_word:LW12
Network 4
LD     SM0.0
A      Sensor_Tow:I1.5
EU
LD     Reset_Tow_HMI:V152.7
LD     Counter_tow:C10
A      Timer_for_not_reset_CNT:T111
A      Sensor_Tow:I1.5
OLD
CTU    Counter_tow:C10, #Tedade_dor_word:LW12
Network 5
LD     Counter_tow:C10
S      Q2.7, 1
Network 6
LD     Q2.7
TON    Time_for_stop_tow:T110, 20
Network 7
LD     Time_for_stop_tow:T110
R      Q2.7, 1
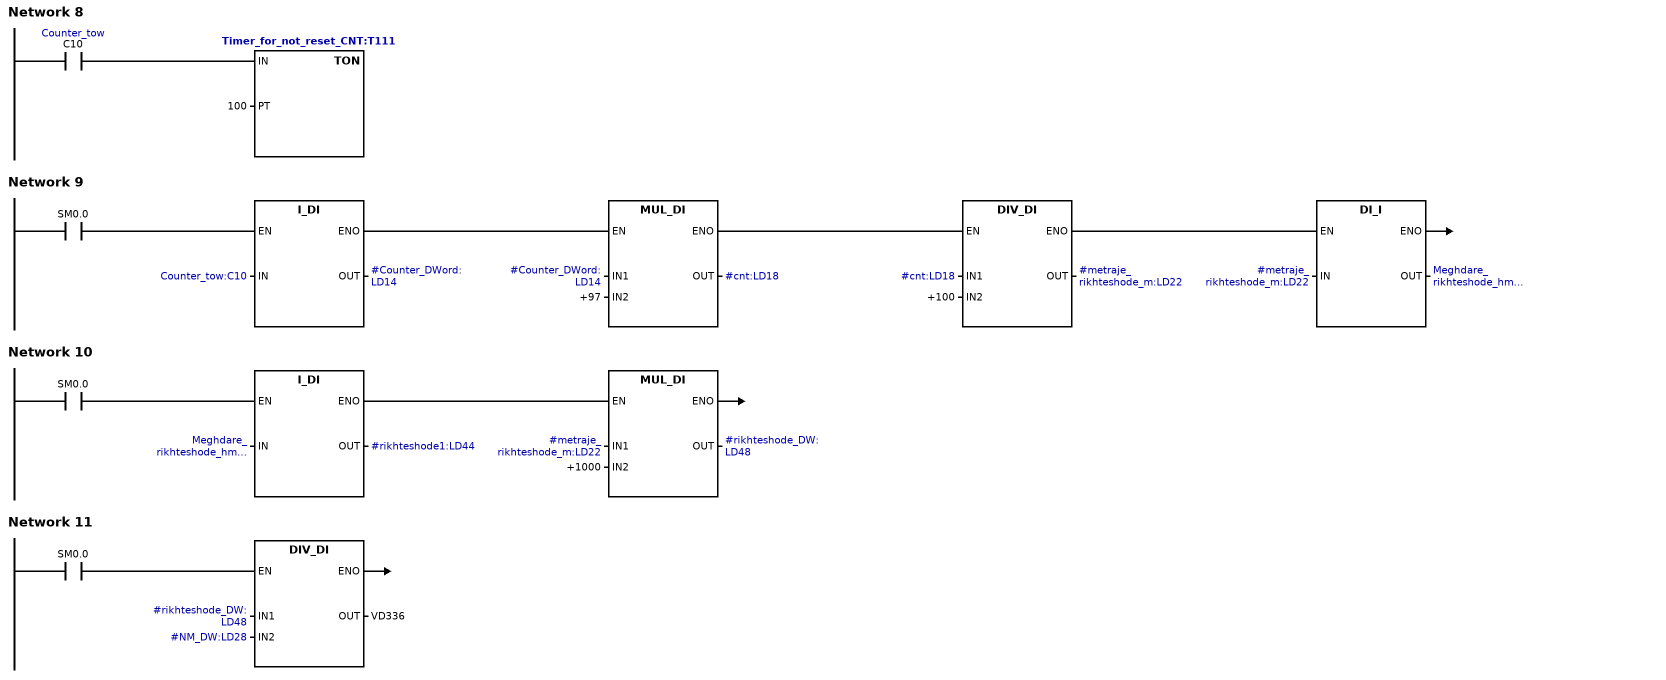
Network 8
LD     Counter_tow:C10
TON    Timer_for_not_reset_CNT:T111, 100
Network 9
LD     SM0.0
ITD    Counter_tow:C10, #Counter_DWord:LD14
AENO
MOVD   #Counter_DWord:LD14, #cnt:LD18
AENO
*D     +97, #cnt:LD18
AENO
MOVD   #cnt:LD18, #metraje_rikhteshode_m:LD22
AENO
/D     +100, #metraje_rikhteshode_m:LD22
AENO
DTI    #metraje_rikhteshode_m:LD22, Meghdare_rikhteshode_hm:VW226
Network 10
LD     SM0.0
ITD    Meghdare_rikhteshode_hm:VW226, #rikhteshode1:LD44
AENO
MOVD   #metraje_rikhteshode_m:LD22, #rikhteshode_DW:LD48
*D     +1000, #rikhteshode_DW:LD48
Network 11
LD     SM0.0
MOVD   #rikhteshode_DW:LD48, VD336
/D     #NM_DW:LD28, VD336
Network 13 // Network Title
// Network Comment
END_SUBROUTINE_BLOCK
